// Mitsubishi GX Works2 project: Traffic light   PLC: FX3U/FX3UC

PROGRAM MAIN
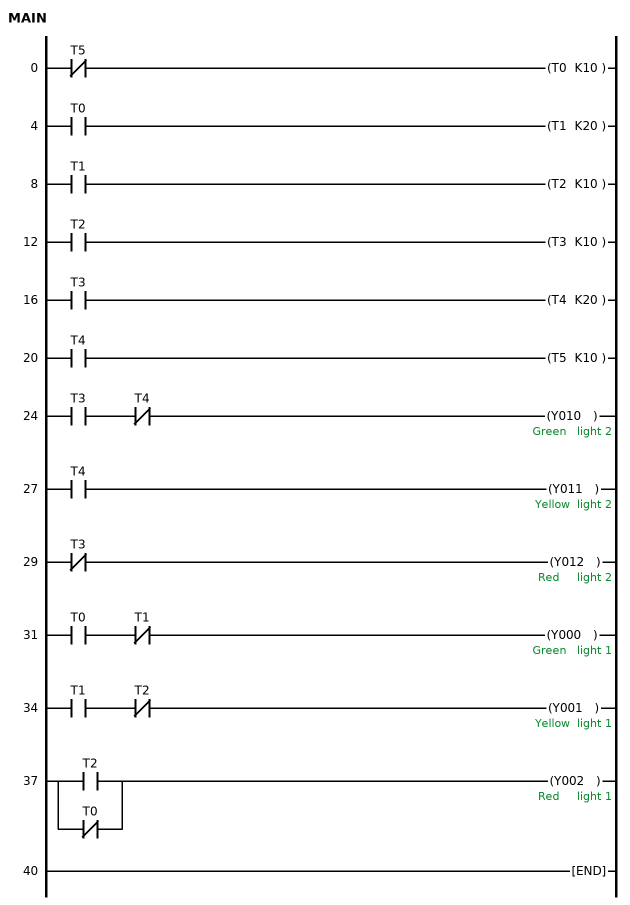
0     LDI     T5
      OUT     T0 K10
4     LD      T0
      OUT     T1 K20
8     LD      T1
      OUT     T2 K10
12    LD      T2
      OUT     T3 K10
16    LD      T3
      OUT     T4 K20
20    LD      T4
      OUT     T5 K10
24    LD      T3
      ANI     T4
      OUT     Y010  ; Green   light 2
27    LD      T4
      OUT     Y011  ; Yellow  light 2
29    LDI     T3
      OUT     Y012  ; Red     light 2
31    LD      T0
      ANI     T1
      OUT     Y000  ; Green   light 1
34    LD      T1
      ANI     T2
      OUT     Y001  ; Yellow  light 1
37    LD      T2
      ORI     T0
      OUT     Y002  ; Red     light 1
40    END
END_PROGRAM
